{attribute 'GeneratedUsingTerminal: KL1202'}
{attribute addProperty BoxType "KL1202"}
{attribute addProperty Description ""}
{attribute addProperty Physics ""}
{attribute addProperty Id "Channel_1AT %Q*Channel_72DF63360Channel_2AT %Q*Channel_72DF63360"}
{attribute addProperty CRC "3968136300"}
{attribute addProperty Size "0"}
TYPE KL1202_EC84F46C :
STRUCT
	{attribute addProperty Name "Channel_1"}
	Channel_1 : Channel_72DF6336;
	{attribute addProperty Name "Channel_2"}
	Channel_2 : Channel_72DF6336;
END_STRUCT
END_TYPE

(* stored: Version 1.2.0.0, ProductVersion 3.1.4024.11
   DUT KL1202_EC84F46C: Id {24ed4785-95b0-4b84-91cf-fe72d9756b85} *)
